SUBAPPLICATION GetEndpointFromOrchestrationHTTPPFull (* Get the endpoint at INDEX from a request orchestration response *)
  (* Standard: 61499-2; Description: Copyright (c) 2019 fortiss GmbH This program and the accompanying materials are made available under the terms of the Eclipse Public License 2.0 which is available at https://www.eclipse.org/legal/epl-2.0/ SPDX-License-Identifier: EPL-2.0 *)
  (* Version 1.0, 2019-02-19, Jose Cabral, fortiss GmbH *)
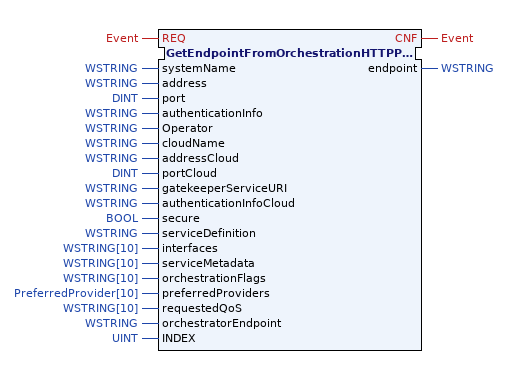
  EVENT_INPUT
    REQ; (* Request orchestration *)
  END_EVENT
  EVENT_OUTPUT
    CNF; (* Request finished *)
  END_EVENT
  VAR_INPUT
    systemName : WSTRING; (* Identification of the system *)
    address : WSTRING; (* Address of the offered services *)
    port : DINT; (* Port of the of the offered services *)
    authenticationInfo : WSTRING; (* Authentication info of the system *)
    Operator : WSTRING; (* Company (the capital  O is to avoid clash when exporting to C++) *)
    cloudName : WSTRING; (* Identification of the cloud *)
    addressCloud : WSTRING; (* Address to access the cloud *)
    portCloud : DINT; (* Port to access the cloud *)
    gatekeeperServiceURI : WSTRING; (* (Unclear documentation) *)
    authenticationInfoCloud : WSTRING; (* Authentication info of the cloud *)
    secure : BOOL; (* (Unclear documentation) *)
    serviceDefinition : WSTRING; (* Identification of the service *)
    interfaces : ARRAY [0..9] OF WSTRING; (* Interfaces implemented by the service *)
    serviceMetadata : ARRAY [0..9] OF WSTRING; (* Metadata of the service in key=value format *)
    orchestrationFlags : ARRAY [0..9] OF WSTRING; (* These flags can be set to tailor the orchestration process (use just the names of the flags to be enabled) *)
    preferredProviders : ARRAY [0..9] OF PreferredProvider; (* There can be a list from the Consumer stating which other Application Systems (even from other Clouds) it wishes to connect. If this field is filled out, the Orchestrator will try to facilitate these preferences *)
    requestedQoS : ARRAY [0..9] OF WSTRING; (* This object will be presenting the Consumer’s selected QoS level. Not implemented *)
    orchestratorEndpoint : WSTRING; (* Enpoint of the orchestrator *)
    INDEX : UINT; (* Position in the array of the requested forms *)
  END_VAR
  VAR_OUTPUT
    endpoint : WSTRING; (* Endpoint at position INDEX from orchestration forms *)
  END_VAR
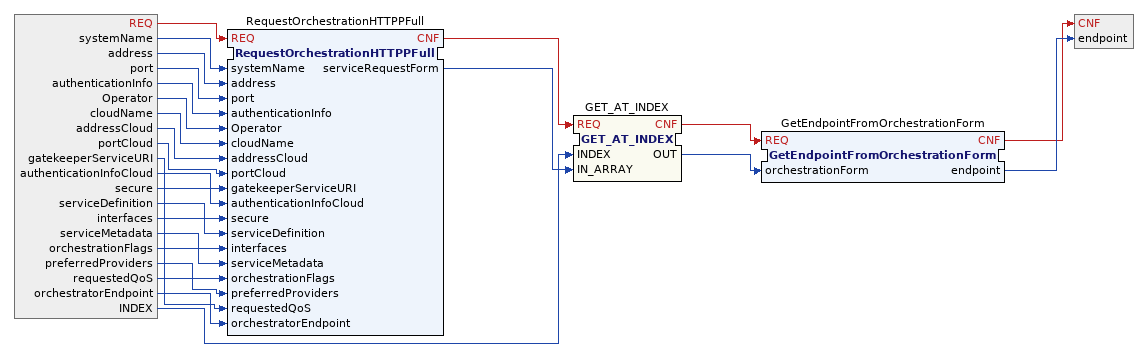
  FBS
    GET_AT_INDEX : GET_AT_INDEX;
  END_FBS
  SUBAPPS
    GetEndpointFromOrchestrationForm : GetEndpointFromOrchestrationForm;
    RequestOrchestrationHTTPPFull : RequestOrchestrationHTTPPFull;
  END_SUBAPPS
  EVENT_CONNECTIONS
    GET_AT_INDEX.CNF TO GetEndpointFromOrchestrationForm.REQ;
    GetEndpointFromOrchestrationForm.CNF TO CNF;
    REQ TO RequestOrchestrationHTTPPFull.REQ;
    RequestOrchestrationHTTPPFull.CNF TO GET_AT_INDEX.REQ;
  END_CONNECTIONS
  DATA_CONNECTIONS
    GET_AT_INDEX.OUT TO GetEndpointFromOrchestrationForm.orchestrationForm;
    INDEX TO GET_AT_INDEX.INDEX;
    GetEndpointFromOrchestrationForm.endpoint TO endpoint;
    systemName TO RequestOrchestrationHTTPPFull.systemName;
    address TO RequestOrchestrationHTTPPFull.address;
    port TO RequestOrchestrationHTTPPFull.port;
    authenticationInfo TO RequestOrchestrationHTTPPFull.authenticationInfo;
    Operator TO RequestOrchestrationHTTPPFull.Operator;
    cloudName TO RequestOrchestrationHTTPPFull.cloudName;
    addressCloud TO RequestOrchestrationHTTPPFull.addressCloud;
    portCloud TO RequestOrchestrationHTTPPFull.portCloud;
    gatekeeperServiceURI TO RequestOrchestrationHTTPPFull.gatekeeperServiceURI;
    authenticationInfoCloud TO RequestOrchestrationHTTPPFull.authenticationInfoCloud;
    secure TO RequestOrchestrationHTTPPFull.secure;
    serviceDefinition TO RequestOrchestrationHTTPPFull.serviceDefinition;
    interfaces TO RequestOrchestrationHTTPPFull.interfaces;
    serviceMetadata TO RequestOrchestrationHTTPPFull.serviceMetadata;
    RequestOrchestrationHTTPPFull.serviceRequestForm TO GET_AT_INDEX.IN_ARRAY;
    preferredProviders TO RequestOrchestrationHTTPPFull.preferredProviders;
    orchestrationFlags TO RequestOrchestrationHTTPPFull.orchestrationFlags;
    requestedQoS TO RequestOrchestrationHTTPPFull.requestedQoS;
    orchestratorEndpoint TO RequestOrchestrationHTTPPFull.orchestratorEndpoint;
  END_CONNECTIONS
END_SUBAPPLICATION
